PROGRAM MAIN
VAR	

END_VAR

	GVL.In := 1;
	GVL.Out := 1;

END_PROGRAM

(* stored: Version 1.1.0.1, ProductVersion 3.1.4024.0
   POU MAIN: Id {cf35716e-8769-4551-8e5a-9323d324a38e}, SpecialFunc None *)
